(* CODESYS project xlh_ha_client_00_05.project
   Author: Pascal Helfenstein
   Title: xlh_ha
   Company: xemax ag

Project tree, tasks and I/O mapping:
  xlh_base : CODESYS Control for Raspberry Pi 64 SL, CODESYS, order no. 2302000009, version 4.18.0.0
    application app
      libraries: Standard, 3.5.18.0 (System); StringUtils, 3.5.20.0 (System); VisuDialogs, * (System); Web Socket Client SL, 1.12.0.0 (CODESYS); Net Base Services, * (3S - Smart Software Solutions GmbH); MQTT Client SL, 1.12.0.0 (CODESYS); Util, 3.5.21.0 (System); String Functions, * (CODESYS); SysTimeRtc, * (System); SysTime, 3.5.17.0 (System); CmpIecTask, * (System); Memory, 3.5.17.0 (3S - Smart Software Solutions GmbH)
      task MainTask (cyclic, interval t#20ms, priority 1) calls LOCAL_TIME_AND_TIME_ZONE, TASK_INFO, io, MAIN
      task VISU_TASK (cyclic, interval 100 ms, priority 31) calls VisuElems.Visu_Prg
      program MAIN [ST]
      program io [ST]
      IoT/
        DEVICES/
          function block _000_FB_VISU_BASE [ST]
          function block _200_FB_DEVICE_SHELLY_BASE [ST]: statusUpdate, startup, newMessage
          function block _202_FB_DEVICE_SHELLY_1PM_TEMP [ST]: newMessage
          interface IDevice
          interface IDeviceZigbee2Mqtt
          interface IDeviceShelly
          function block _201_FB_DEVICE_SHELLY_1PM_PLUG [ST]: publisher, newMessage
          function block _300_FB_DEVICE_ZIGBEE2MQTT_BASE [ST]: statusUpdate, startup, newMessage
          VISU/
            visualisation VISU_FB_DEVICE_SHELLY_RELAIS
            visualisation VISU_FB_DEVICE_SHELLY_RELAIS_TEMP
          function block _100_FB_DEVICE [ST]: subscriber, publisher, startup, popFifoPublish, newMessage, statusUpdate, pushFifoPublish
          trace Trace (task MainTask): io.fbShellyPlug2._fbMqttPublisher.xBusy, io.fbShellyPlug2._fbMqttPublisher.xDone, io.fbShellyPlug2._fbMqttPublisher.xExecute, io.fbShellyPlug2._iFifoPopCycleCounter
          interface IVisu
        MQTT_Client/
          function TERMINATE_STRING [ST]
          function block FB_MQTT_CLIENT [ST]: pMqttClient
          function GET_VALUE_FROM_MSG [ST]
          function GET_REAL_FROM_VALUE [ST]
          function GET_BOOL_FROM_VALUE [ST]
          function GET_INT_FROM_VALUE [ST]
          function GET_STRING_FROM_VALUE [ST]
          function GET_LREAL_FROM_VALUE [ST]
        global variables GC
        program TASK_INFO [ST]
        program LOCAL_TIME_AND_TIME_ZONE [ST]
      visualisation VISUALIZATION
    SoftMotion General Axis Pool
    GPIOs_A_B : GPIOs A/B, CODESYS, version 4.18.0.0
        unmapped channels: digital inputs (GPIO0..GPIO31), digital outputs (GPIO0..GPIO31)
    Onewire
    Camera device
      <Empty>
    SPI
    I²C
  libraries: VisuSymbols, 4.5.0.0 (System)
  text list GlobalTextList
  5ce3da45-db07-42e7-a21c-a00fff4ed8f6|C:\Users\a.werner\Documents\background.jpg
*)

// xlh_base/app/IoT/GC
{attribute 'qualified_only'}
VAR_GLOBAL CONSTANT
	//STRING_SIZE: INT := 255;
	STRING_SIZE_TOPIC: INT := 1024;
	STRING_SIZE_MESSAGE_TX: INT := 1024;
	STRING_SIZE_MESSAGE_RX: INT := 2048;
END_VAR

// xlh_base/app/IoT/LOCAL_TIME_AND_TIME_ZONE
PROGRAM LOCAL_TIME_AND_TIME_ZONE
VAR_OUTPUT
	stUTC_Timestamp : SysTime;
	stCTE_Timestamp : SysTime;
	stJoinedTimestamp : SysTime;
	stCombinedTimestamp : SysTime;
	uiYear : YEAR; (* 1970..2106 *)
    uiMonth : MONTH;
    uiDay : DAY;
    uiHour : UINT;
    uiMinute : UINT;
    uiSecond : UINT;
    uiMilliseconds : MILLISECOND;
    eWeekday : WEEKDAY;
    datDate : DATE;
    todTime : TIME_OF_DAY;
	eError : Util.ERROR;
	xLeapYear : BOOL;
END_VAR
VAR CONSTANT
    /// Coordinated Universal Time
    gc_tzTimeZoneUTC : TimeZone := (asgPeriod := [(sName:='UTC')]);

    /// Central Europe Time
    gc_tzTimeZoneCET : TimeZone :=
    (
        iBias := 60 (* T#1M => minutes *),
        asgPeriod := [
        ( (* (CEST -> CET) - Last Sunday in Oktober at 03:00:00.000 (CEST) *)
            sName:='CET',
            dtDate := (uiMonth := 10, eWeekday := WEEKDAY.SUNDAY, uiDay := 5, uiHour := 3)
        ),( (* (CET -> CEST) - Last Sunday in March at 02:00:00.000 (CET) *)
            sName := 'CEST',
            dtDate := (uiMonth := 3, eWeekday := WEEKDAY.SUNDAY, uiDay := 5, uiHour := 2),
            iBias := 60 (* T#1M => minutes *)
        )]
    );
END_VAR

SysTimeRtcHighResGet(pTimestamp := stUTC_Timestamp);
// Conversion from UTC timestamp (e.g. from SysTimeRtcHighResGet) to the current period and the local date and time related to the TimeZone parameter.
stCTE_Timestamp := Util.LocalDateTime(	tzTimeZone := gc_tzTimeZoneCET, 
										uliDateTime := stUTC_Timestamp,
										eErrorID => eError);

// Splitting a timestamp into the components of a point in time.
eError := Util.SplitDateTime(	uliDateTime := stCTE_Timestamp,
				uiYear => uiYear,
				uiMonth =>  uiMonth,
				uiDay => uiDay,
				uiHour => uiHour,
				uiMinute => uiMinute,
				uiSecond =>  uiSecond,
				uiMilliseconds => uiMilliseconds,
				eWeekday => eWeekday);

// Joining the components of a point in time to a timestamp (UTC). 
stJoinedTimestamp :=  Util.JoinDateTime( 	uiYear := uiYear,
									uiMonth :=  uiMonth,
									uiDay := uiDay,
									uiHour := uiHour,
									uiMinute := uiMinute,
									uiSecond :=  uiSecond,
									uiMilliseconds := uiMilliseconds);
									
// Separates a timestamp in its IEC data typed parts.
 Util.SeparateDateTime(	uliDateTime := stCTE_Timestamp,
    				eWeekDay => eWeekDay,
    				datDate => datDate,
    				todTime => todTime);
					
// Combines the IEC data typed parts to a timestamp.
stCombinedTimestamp := Util.CombineDateTime(	datDate := datDate, 
												todTime := todTime, 
												eErrorID => eError);
						
// Calculates the appropriate value of the WEEKDAY enum that matches the parameter datDate.
eWeekday := Util.DayOfWeek(	datDate := datDate, 
							eErrorID => eError);

// Checks whether the year (uiYear) passed represents a leap year.					
xLeapYear := Util.IsLeapYear(	uiYear := uiYear,
								eErrorID => eError);

END_PROGRAM

// xlh_base/app/IoT/TASK_INFO
PROGRAM TASK_INFO
VAR
    Result: CmpIecTask.RTS_IEC_RESULT;
    hCurrentTask : CmpIecTask.RTS_IEC_HANDLE;
    pCurrentTaskInfo: POINTER TO Task_Info2;
    stCurrentTaskInfo: Task_Info2;
END_VAR
VAR_OUTPUT
	fCycleTime: LREAL;
	fInterval: LREAL;
	fCycleTimeUs: LREAL;
	fJitterUs: LREAL;
	fJitterOffsetInterwalUs: LREAL;
END_VAR

// https://content.helpme-codesys.com/en/libs/CmpIecTask/Current/index.html
// https://forge.codesys.com/forge/talk/Engineering/thread/b7e9b2b353/
// https://medium.com/@sean.gongz/how-to-get-current-task-actual-cycle-time-in-codesys-267384bcd3b7

hCurrentTask := IecTaskGetCurrent(pResult:=ADR(Result));
pCurrentTaskInfo := IecTaskGetInfo3(hIecTask:=hCurrentTask, pResult:=ADR(Result));
stCurrentTaskInfo := pCurrentTaskInfo^;

fCycleTimeUs := TO_LREAL(TO_DINT(stCurrentTaskInfo.dwInterval) + stCurrentTaskInfo.iJitter);
fInterval := TO_LREAL(stCurrentTaskInfo.dwInterval);
fJitterUs := TO_LREAL(stCurrentTaskInfo.iJitter);
fJitterOffsetInterwalUs := fInterval + fJitterUs;
fCycleTime := fCycleTimeUs / 1000000.0;

END_PROGRAM

// xlh_base/app/io
PROGRAM io
VAR_INPUT
	fbShellyPlug1: _201_FB_DEVICE_SHELLY_1PM_PLUG := (bEnable:=TRUE, sMqttTopicBase:='shellyplug-81', sLabel:='shellyplug-81');
	fbShellyPlug2: _201_FB_DEVICE_SHELLY_1PM_PLUG := (bEnable:=TRUE, sMqttTopicBase:='shellyplug-82', sLabel:='shellyplug-82');
	fbShellyPm1: _201_FB_DEVICE_SHELLY_1PM_PLUG := (bEnable:=FALSE, sMqttTopicBase:='shellyplus1pm-88', sLabel:='shellyplus1pm-88');
	fbShellyPm2: _202_FB_DEVICE_SHELLY_1PM_TEMP := (bEnable:=TRUE, sMqttTopicBase:='shellyplus1pm-51', sLabel:='shellyplus1pm-51');
END_VAR
VAR
	_bStartup: BOOL := TRUE;
	_aIoClients: ARRAY [0..(iNR_OF_IO_CLIENTS-1)] OF POINTER TO _100_FB_DEVICE;
	_fbMqttClient: FB_MQTT_CLIENT := (sClientId:='xlh_base_ha_io');
	_iI: INT;
	//
	_bDummy: BOOL;
END_VAR
VAR CONSTANT
	iNR_OF_IO_CLIENTS: INT := 20;
END_VAR

IF _bStartup THEN
	_bStartup := FALSE;
	_aIoClients[_iI] := ADR(fbShellyPlug1); _iI := _iI + 1;
	_aIoClients[_iI] := ADR(fbShellyPlug2); _iI := _iI + 1;
	_aIoClients[_iI] := ADR(fbShellyPm1); _iI := _iI + 1;
	_aIoClients[_iI] := ADR(fbShellyPm2); _iI := _iI + 1;
	
	FOR _iI := 0 TO (iNR_OF_IO_CLIENTS-1) BY 1 DO
		IF (_aIoClients[_iI] > 16#0) THEN
			_aIoClients[_iI]^.pMqttClient := ADR(_fbMqttClient);
			_aIoClients[_iI]^.startup();	
		END_IF
	END_FOR	
	
	_fbMqttClient.bEnable := TRUE;
END_IF

_fbMqttClient();

FOR _iI := 0 TO (iNR_OF_IO_CLIENTS-1) BY 1 DO
	IF (_aIoClients[_iI] >16#0) THEN
		_aIoClients[_iI]^();	
	END_IF
END_FOR

_bDummy := _fbMqttClient.bConnected;

END_PROGRAM

// xlh_base/app/IoT/DEVICES/_201_FB_DEVICE_SHELLY_1PM_PLUG
FUNCTION_BLOCK _201_FB_DEVICE_SHELLY_1PM_PLUG EXTENDS _200_FB_DEVICE_SHELLY_BASE
VAR_INPUT
	bRelais: BOOL;
	bResetEnergy: BOOL;
END_VAR
VAR_OUTPUT
	bRelaisState: BOOL;
	fVoltage: LREAL;
	fCurrent: LREAL;
	fPower: LREAL;
	fElectricalEnergy: LREAL;
END_VAR
VAR
	//
	_fbRtRelais: R_TRIG;
	_fbFtRelais: F_tRIG;
	_fbTonDiffRelaisState: TON;
END_VAR
VAR CONSTANT
	_tACTION_TIME_NOT_EQUAL: TIME := T#500MS;
END_VAR

SUPER^();
IF bResetEnergy THEN
	fElectricalEnergy := 0.0;
ELSE
	fElectricalEnergy := fElectricalEnergy + fPower * TASK_INFO.fCycleTime;
END_IF

METHOD publisher : BOOL
VAR_INPUT
END_VAR

VAR
	bPublish: BOOL;
	sPublishMessage : STRING(GC.STRING_SIZE_MESSAGE_TX);
END_VAR
THIS^._fbTonDiffRelaisState(IN:=((THIS^.bRelais <> THIS^.bRelaisState) AND NOT _fbTonDiffRelaisState.Q), PT:=THIS^._tACTION_TIME_NOT_EQUAL);
THIS^._fbRtRelais(CLK:=THIS^.bRelais);
THIS^._fbFtRelais(CLK:=THIS^.bRelais);
bPublish := _fbTonDiffRelaisState.Q OR _fbRtRelais.Q OR _fbFtRelais.Q;

IF bPublish THEN
	sPublishMessage := '{"id":1, "src":"';
	Stu.StrConcatA(pstFrom:=ADR(THIS^.sMqttTopicBase), pstTo:=ADR(sPublishMessage), iBufferSize:=GC.STRING_SIZE_MESSAGE_TX);
	Stu.StrConcatA(pstFrom:=ADR('/relais", "method":"Switch.Set", "params":{"id":0, "on":'), pstTo:=ADR(sPublishMessage), iBufferSize:=GC.STRING_SIZE_MESSAGE_TX);
	//sPublishMessage := CONCAT(sPublishMessage, THIS^.sMqttTopicBase);
	//sPublishMessage := CONCAT(sPublishMessage, '/relais", "method":"Switch.Set", "params":{"id":0, "on":');
	IF THIS^.bRelais THEN
		Stu.StrConcatA(pstFrom:=ADR('true}}'), pstTo:=ADR(sPublishMessage), iBufferSize:=GC.STRING_SIZE_MESSAGE_TX);
		//sPublishMessage := CONCAT(sPublishMessage, 'true}}');
	ELSE
		Stu.StrConcatA(pstFrom:=ADR('false}}'), pstTo:=ADR(sPublishMessage), iBufferSize:=GC.STRING_SIZE_MESSAGE_TX);
		//sPublishMessage := CONCAT(sPublishMessage, 'false}}');
	END_IF
	THIS^.pushFifoPublish(THIS^._wsPublishTopic, sPublishMessage);
END_IF

SUPER^.publisher();
END_METHOD

METHOD newMessage : BOOL
VAR_INPUT
	
END_VAR
VAR

	
END_VAR
SUPER^.newMessage();
IF (_fbMqttSubscriber.wsLastTopic = _wsMqttTopicEvent) OR
   (_fbMqttSubscriber.wsLastTopic = _wsMqttTopicStatus) THEN
	bRelaisState := GET_BOOL_FROM_VALUE(bRelaisState, GET_VALUE_FROM_MSG('output', ADR(_sSubscribedMessage)));
	fVoltage := GET_LREAL_FROM_VALUE(fVoltage, GET_VALUE_FROM_MSG('voltage', ADR(_sSubscribedMessage)));
	fCurrent := GET_LREAL_FROM_VALUE(fCurrent, GET_VALUE_FROM_MSG('current', ADR(_sSubscribedMessage)));
	fPower := GET_LREAL_FROM_VALUE(fPower, GET_VALUE_FROM_MSG('apower', ADR(_sSubscribedMessage)));
		
END_IF
IF (_fbMqttSubscriber.wsLastTopic = _wsMqttTopicStatus) THEN
	sSsid := GET_STRING_FROM_VALUE(sSsid, GET_VALUE_FROM_MSG('ssid', ADR(_sSubscribedMessage)));
	sMacId := GET_STRING_FROM_VALUE(sSsid, GET_VALUE_FROM_MSG('bssid', ADR(_sSubscribedMessage)));	
END_IF

(*
// FixMe: total energy from status Message

Topic: shellyplus1pm-51/status/rpcQoS: 0

{"id":1,"src":"shellyplus1pm-e465b8b7ad64","dst":"shellyplus1pm-51/status","result":{"ble":{},"cloud":{"connected":false},"input:0":
{"id":0,"state":false},"mqtt":{"connected":true},
"switch:0":{"id":0, "source":"MQTT", "output":false, "apower":0.0, "voltage":236.0, "current":0.000, 
"aenergy":{"total":2431.000,"by_minute":[0.000,0.000,0.000],"minute_ts":1765258740},
"temperature":{"tC":38.2, "tF":100.8}},"sys":{"mac":"E465B8B7AD64","restart_required":false,"time":"06:39","unixtime":1765258775,"last_sync_ts":1765258399,"uptime":380,"ram_size":250884,"ram_free":138740,"ram_min_free":127852,"fs_size":393216,"fs_free":126976,"cfg_rev":40,"kvs_rev":0,"schedule_rev":1,"webhook_rev":0,"btrelay_rev":0,"available_updates":{},"reset_reason":1,"utc_offset":3600},"temperature:100":{"id": 100,"tC":20.1, "tF":68.1},"temperature:101":{"id": 101,"tC":19.9, "tF":67.9},"temperature:102":{"id": 102,"tC":20.0, "tF":68.0},"wifi":{"sta_ip":"192.168.1.51","status":"got ip","ssid":"hpna_fritz_box","bssid":"3c:37:12:6b:47:96","rssi":-28},"ws":{"connected":false}}}
*)
END_METHOD

END_FUNCTION_BLOCK

// xlh_base/app/IoT/DEVICES/_200_FB_DEVICE_SHELLY_BASE
FUNCTION_BLOCK _200_FB_DEVICE_SHELLY_BASE EXTENDS _100_FB_DEVICE IMPLEMENTS IDeviceShelly
VAR_INPUT
END_VAR
VAR_OUTPUT
	fTemperaturePcb: LREAL;
	sSsid: STRING(255);
	sMacId: STRING(255);
	iRssi: INT;
END_VAR
VAR
	//
	_wsMqttTopicEvent: WSTRING(GC.STRING_SIZE_TOPIC);
	_wsMqttTopicStatus: WSTRING(GC.STRING_SIZE_TOPIC);
	_fTimer: LREAL := 0.0;
END_VAR
VAR CONSTANT
	_fREFRESH_TIME: LREAL := 300.0;
END_VAR

SUPER^();

_fTimer := LIMIT(0.0, _fTimer + TASK_INFO.fCycleTime, 99999.0);
IF _fTimer >= _fREFRESH_TIME THEN
	_fTimer := 0.0;
	statusUpdate();
END_IF

METHOD statusUpdate : BOOL
VAR_INPUT
END_VAR
VAR
	sPublishMessage : STRING(GC.STRING_SIZE_MESSAGE_TX);
END_VAR
SUPER^.statusUpdate();
sPublishMessage := '{"id":1, "src":"';
Stu.StrConcatA(pstFrom:=ADR(THIS^.sMqttTopicBase), pstTo:=ADR(sPublishMessage), iBufferSize:=GC.STRING_SIZE_MESSAGE_TX);
Stu.StrConcatA(pstFrom:=ADR('/status", "method":"Shelly.GetStatus"}'), pstTo:=ADR(sPublishMessage), iBufferSize:=GC.STRING_SIZE_MESSAGE_TX);
//sPublishMessage := CONCAT(sPublishMessage, THIS^.sMqttTopicBase);
//sPublishMessage := CONCAT(sPublishMessage, '/status", "method":"Shelly.GetStatus"}');
THIS^.pushFifoPublish(THIS^._wsPublishTopic, sPublishMessage);
END_METHOD

METHOD startup : BOOL
VAR_INPUT
END_VAR

VAR
END_VAR
SUPER^.startup();

_wsPublishTopic := "";
Stu.StrConcatW(pstFrom:=ADR(_wsMqttTopicBase), pstTo:=ADR(_wsPublishTopic), iBufferSize:=GC.STRING_SIZE_TOPIC);
Stu.StrConcatW(pstFrom:=ADR("/rpc"), pstTo:=ADR(_wsPublishTopic), iBufferSize:=GC.STRING_SIZE_TOPIC);

_wsMqttTopicEvent := "";
Stu.StrConcatW(pstFrom:=ADR(_wsMqttTopicBase), pstTo:=ADR(_wsMqttTopicEvent), iBufferSize:=GC.STRING_SIZE_TOPIC);
Stu.StrConcatW(pstFrom:=ADR("/events/rpc"), pstTo:=ADR(_wsMqttTopicEvent), iBufferSize:=GC.STRING_SIZE_TOPIC);
		
_wsMqttTopicStatus := "";
Stu.StrConcatW(pstFrom:=ADR(_wsMqttTopicBase), pstTo:=ADR(_wsMqttTopicStatus), iBufferSize:=GC.STRING_SIZE_TOPIC);
Stu.StrConcatW(pstFrom:=ADR("/status/rpc"), pstTo:=ADR(_wsMqttTopicStatus), iBufferSize:=GC.STRING_SIZE_TOPIC);
END_METHOD

METHOD newMessage : BOOL
VAR_INPUT
	
END_VAR
VAR

	
END_VAR
SUPER^.newMessage();
IF (_fbMqttSubscriber.wsLastTopic = _wsMqttTopicEvent) OR
   (_fbMqttSubscriber.wsLastTopic = _wsMqttTopicStatus) THEN
   fTemperaturePcb := GET_LREAL_FROM_VALUE(fTemperaturePcb, GET_VALUE_FROM_MSG('temperature":{"tC', ADR(_sSubscribedMessage)));
	iRssi := GET_INT_FROM_VALUE(iRssi, GET_VALUE_FROM_MSG('rssi', ADR(_sSubscribedMessage)));	
END_IF
IF (_fbMqttSubscriber.wsLastTopic = _wsMqttTopicStatus) THEN
	sSsid := GET_STRING_FROM_VALUE(sSsid, GET_VALUE_FROM_MSG('ssid', ADR(_sSubscribedMessage)));
	sMacId := GET_STRING_FROM_VALUE(sSsid, GET_VALUE_FROM_MSG('bssid', ADR(_sSubscribedMessage)));	
END_IF
END_METHOD

END_FUNCTION_BLOCK

// xlh_base/app/IoT/DEVICES/_100_FB_DEVICE
FUNCTION_BLOCK _100_FB_DEVICE EXTENDS _000_FB_VISU_BASE IMPLEMENTS IDevice
VAR_INPUT
	bEnable: BOOL;
	sMqttTopicBase: STRING(255);
	pMqttClient: POINTER TO FB_MQTT_CLIENT;
END_VAR
VAR
	_wsMqttTopicBase: WSTRING(GC.STRING_SIZE_TOPIC);
	//
	_fbRtMqttClientConnected: R_TRIG;
	_fbFtMqttClientConnected: F_TRIG;
	_fbRtMqttSubscriberActive: R_TRIG;
	_fbFtMqttSubscriberActive: F_TRIG;
	_fbRtError: R_TRIG;
	_fbTonConnect: TON;
	_fbTonDisconnect: TON;
	//
	_fbMqttSubscriber : MQTT.MQTTSubscribe;
	_wsSubcribedTopicFilter : WSTRING(GC.STRING_SIZE_TOPIC);
	_sSubscribedMessage : STRING(GC.STRING_SIZE_MESSAGE_RX);	
	//
	_fbMqttPublisher : MQTT.MQTTPublish;
	_wsPublishTopic : WSTRING(GC.STRING_SIZE_TOPIC);
	_sPublishMessage : STRING(GC.STRING_SIZE_MESSAGE_TX);
	//
	_iFifoPos: INT;
	_iFifoPosMax: INT;
	_awsPublishTopic: ARRAY[0..(_iFIFO_SIZE-1)] OF WSTRING(GC.STRING_SIZE_TOPIC);
	_asPublishMessage: ARRAY[0..(_iFIFO_SIZE-1)] OF STRING(GC.STRING_SIZE_MESSAGE_TX);
	_iFifoPopCycleCounter: INT;
	//
	_todMessageUpdate: TIME_OF_DAY;
END_VAR
VAR CONSTANT
	_iFIFO_SIZE: INT := 25;
	_iFIFO_DELAY_COUNTER: INT := 5;
END_VAR

THIS^.subscriber();
THIS^.publisher();

METHOD subscriber : BOOL
VAR_INPUT
END_VAR
THIS^._fbRtMqttClientConnected(CLK:=THIS^.pMqttClient^.bConnected);
THIS^._fbFtMqttClientConnected(CLK:=THIS^.pMqttClient^.bConnected);
THIS^._fbRtError(CLK:=THIS^.pMqttClient^.bError);
IF THIS^._fbRtMqttClientConnected.Q THEN
	THIS^._fbMqttSubscriber.xEnable := TRUE;
END_IF
IF THIS^._fbRtError.Q OR THIS^._fbFtMqttClientConnected.Q THEN
	THIS^._fbMqttSubscriber.xEnable := FALSE;
END_IF
THIS^._fbTonDisconnect.IN := THIS^.pMqttClient^.bConnected AND THIS^._fbMqttSubscriber.xEnable AND NOT THIS^._fbMqttSubscriber.xBusy;
THIS^._fbTonDisconnect(PT:=T#3000MS);
IF THIS^._fbTonDisconnect.Q THEN
	THIS^._fbMqttSubscriber.xEnable := FALSE;
END_IF
THIS^._fbTonConnect.IN := THIS^.pMqttClient^.bConnected AND NOT THIS^._fbMqttSubscriber.xEnable;
THIS^._fbTonConnect(PT:=T#500MS);
IF THIS^._fbTonConnect.Q THEN
	THIS^._fbMqttSubscriber.xEnable := TRUE;
END_IF
IF NOT THIS^.bEnable THEN
	THIS^._fbMqttSubscriber.xEnable := FALSE;
END_IF

THIS^._fbMqttSubscriber(mqttClient:=THIS^.pMqttClient^.fbMqttClient,
				wsTopicFilter:=THIS^._wsSubcribedTopicFilter,
		        pbPayload:=ADR(THIS^._sSubscribedMessage),
				udiMaxPayloadSize:=SIZEOF(THIS^._sSubscribedMessage));
TERMINATE_STRING(psIn:=ADR(THIS^._sSubscribedMessage), THIS^._fbMqttSubscriber.udiPayloadSize);

IF THIS^._fbMqttSubscriber.xReceived THEN
	THIS^.newMessage();
END_IF 

THIS^._fbRtMqttSubscriberActive(CLK:=THIS^._fbMqttSubscriber.xSubscribeActive);
THIS^._fbFtMqttSubscriberActive(CLK:=THIS^._fbMqttSubscriber.xSubscribeActive);
IF THIS^._fbRtMqttSubscriberActive.Q THEN
	THIS^.statusUpdate();
END_IF
			
_bDummy := THIS^._fbMqttSubscriber.xEnable;				
_bDummy := THIS^._fbMqttSubscriber.xDone;
_bDummy := THIS^._fbMqttSubscriber.xBusy;
_bDummy := THIS^._fbMqttSubscriber.xError;
_bDummy := THIS^._fbMqttSubscriber.xSubscribeActive;
_wsDummy := THIS^._fbMqttSubscriber.wsLastTopic;
_sDummy := THIS^._sSubscribedMessage;
END_METHOD

METHOD publisher : BOOL
VAR_INPUT

END_VAR
IF THIS^.bEnable THEN
	IF NOT THIS^._fbMqttPublisher.xExecute AND NOT THIS^._fbMqttPublisher.xBusy  THEN
		THIS^._fbMqttPublisher.xExecute := popFifoPublish();  
	END_IF
ELSE
	THIS^._fbMqttPublisher.xExecute := FALSE;
END_IF

THIS^._fbMqttPublisher(mqttClient:=THIS^.pMqttClient^.fbMqttClient, 	 
					   wsTopicName:=_wsPublishTopic,
					   udiTimeOut:=10000,
					   pbPayload:=ADR(_sPublishMessage),
					   udiPayloadSize:=DINT_TO_UDINT(Stu.StrLenA(ADR(_sPublishMessage))));

IF NOT THIS^._fbMqttPublisher.xBusy or THIS^._fbMqttPublisher.xError THEN
	THIS^._fbMqttPublisher.xExecute := FALSE;  
END_IF
END_METHOD

METHOD startup : BOOL
VAR_INPUT
END_VAR

VAR
END_VAR
_wsMqttTopicBase := STRING_TO_WSTRING(sMqttTopicBase);

_wsSubcribedTopicFilter := "";
Stu.StrConcatW(pstFrom:=ADR(_wsMqttTopicBase), pstTo:=ADR(_wsSubcribedTopicFilter), iBufferSize:=GC.STRING_SIZE_TOPIC);
Stu.StrConcatW(pstFrom:=ADR("/#"), pstTo:=ADR(_wsSubcribedTopicFilter), iBufferSize:=GC.STRING_SIZE_TOPIC);
END_METHOD

METHOD popFifoPublish : BOOL
VAR_INPUT

END_VAR
VAR
	iI: INT;
END_VAR
IF _iFifoPos > 0  AND _iFifoPopCycleCounter = 0 THEN
	_iFifoPos := _iFifoPos - 1;
	//MEM.MemFill(ADR(sPublishTopic), INT_TO_UINT(SIZEOF(sPublishTopic)), 16#00);
	//MEM.MemFill(ADR(sPublishMessage), INT_TO_UINT(SIZEOF(sPublishMessage)), 16#00);	
	MEM.MemMove(ADR(_awsPublishTopic[0]), ADR(_wsPublishTopic), SIZEOF(_wsPublishTopic));
	MEM.MemMove(ADR(_asPublishMessage[0]), ADR(_sPublishMessage), SIZEOF(_sPublishMessage));
	FOR iI := 1 TO (_iFIFO_SIZE-1) BY 1 DO
		MEM.MemMove(ADR(_awsPublishTopic[iI]), ADR(_awsPublishTopic[iI-1]), SIZEOF(_awsPublishTopic[iI-1]));
		MEM.MemMove(ADR(_asPublishMessage[iI]), ADR(_asPublishMessage[iI-1]), SIZEOF(_asPublishMessage[iI-1]));
	END_FOR 
	MEM.MemFill(ADR(_awsPublishTopic[_iFIFO_SIZE-1]), SIZEOF(_awsPublishTopic[_iFIFO_SIZE-1]), 16#00);
	MEM.MemFill(ADR(_asPublishMessage[_iFIFO_SIZE-1]), SIZEOF(_asPublishMessage[_iFIFO_SIZE-1]), 16#00);
	
	_iFifoPopCycleCounter := _iFIFO_DELAY_COUNTER;
	popFifoPublish := TRUE;
ELSE
	IF _iFifoPopCycleCounter > 0 THEN
		_iFifoPopCycleCounter := _iFifoPopCycleCounter - 1;
	END_IF
	popFifoPublish := FALSE;	
END_IF
END_METHOD

METHOD newMessage : BOOL
VAR_INPUT
	
END_VAR
VAR

	
END_VAR
THIS^._todMessageUpdate := LOCAL_TIME_AND_TIME_ZONE.todTime;
END_METHOD

METHOD statusUpdate : BOOL
VAR_INPUT
END_VAR

VAR
END_VAR
END_METHOD

METHOD pushFifoPublish : BOOL
VAR_INPUT
	wsTopic: WSTRING(GC.STRING_SIZE_TOPIC);
	sMessage: STRING(GC.STRING_SIZE_MESSAGE_TX);
END_VAR
VAR
	iI: INT;
END_VAR
IF THIS^.bEnable AND _iFifoPos < (_iFIFO_SIZE-1) THEN
	_iFifoPos := _iFifoPos + 1;
	FOR iI := (_iFIFO_SIZE-2) TO 0 BY -1 DO
		MEM.MemMove(ADR(_awsPublishTopic[iI]), ADR(_awsPublishTopic[iI+1]), SIZEOF(_awsPublishTopic[iI+1]));
		MEM.MemMove(ADR(_asPublishMessage[iI]), ADR(_asPublishMessage[iI+1]), SIZEOF(_asPublishMessage[iI+1]));
	END_FOR 
	MEM.MemFill(ADR(_awsPublishTopic[0]), SIZEOF(_awsPublishTopic[0]), 16#00);
	MEM.MemMove(ADR(wsTopic), ADR(_awsPublishTopic[0]), SIZEOF(wsTopic));
	TERMINATE_STRING(psIn:=ADR(_awsPublishTopic[0]), udiLength:=SIZEOF(wsTopic)-1);
	
	MEM.MemFill(ADR(_asPublishMessage[0]), SIZEOF(_asPublishMessage[0]), 16#00);
	MEM.MemMove(ADR(sMessage), ADR(_asPublishMessage[0]), SIZEOF(sMessage));
	TERMINATE_STRING(psIn:=ADR(_asPublishMessage[0]), udiLength:=SIZEOF(sMessage)-1);
	
	pushFifoPublish := TRUE;
ELSE
	pushFifoPublish := FALSE;	
END_IF

IF _iFifoPos > _iFifoPosMax THEN
	_iFifoPosMax := _iFifoPos;
END_IF
END_METHOD

END_FUNCTION_BLOCK

// xlh_base/app/IoT/DEVICES/_000_FB_VISU_BASE
FUNCTION_BLOCK _000_FB_VISU_BASE IMPLEMENTS IVisu
VAR_INPUT
	sLabel: STRING(255) := '';
END_VAR
VAR
	//_bVisuFramShow: BOOL;
	//_iVisuFrame: INT;	
	//_tonVisuFrameShow: TON;
	_bDummy: BOOL;
	_iDummy: INT;
	_rDummy: REAL;
	_fDummy: LREAL;
	_sDummy: STRING(GC.STRING_SIZE_MESSAGE_RX);
	_wsDummy: WSTRING(GC.STRING_SIZE_TOPIC);
END_VAR

(*
_tonVisuFrameShow(IN:=_bVisuFramShow, PT:=T#300S);
IF _tonVisuFrameShow.Q THEN
	_bVisuFramShow := FALSE;
	_iVisuFrame := 0;
END_IF
*)

END_FUNCTION_BLOCK

// xlh_base/app/IoT/DEVICES/IVisu
INTERFACE IVisu

END_INTERFACE

// xlh_base/app/IoT/DEVICES/IDevice
INTERFACE IDevice

END_INTERFACE

// xlh_base/app/IoT/MQTT_Client/FB_MQTT_CLIENT
FUNCTION_BLOCK FB_MQTT_CLIENT
VAR_INPUT
	bEnable: BOOL;
	sHostname: STRING(255) := 'localhost';	
	sClientId: STRING(255) := 'xLH_mqtt_codesys';	
END_VAR
VAR_OUTPUT
	bConnected: BOOL;
	bError: BOOL;
	fbMqttClient : MQTT.MQTTClient := (uiPort:=1883, eMQTTVersion:=MQTT.MQTT_VERSION.V3_1_1, eCommunicationMode:= MQTT.COMMUNICATION_MODE.TCP);
END_VAR
VAR
	_refMqttClient: REFERENCE TO MQTT.MQTTClient;
	_bStartup: BOOL := TRUE;
END_VAR

IF _bStartup THEN
	_bStartup := FALSE;
	_refMqttClient REF= fbMqttClient;
END_IF
fbMqttClient.xEnable := bEnable AND NOT fbMqttClient.xError;
fbMqttClient.sClientId := sClientId;
fbMqttClient(sHostname:=sHostname);
bConnected := fbMqttClient.xConnectedToBroker;
bError := fbMqttClient.xError;

PROPERTY pMqttClient : POINTER TO FB_MQTT_CLIENT
GET
pMqttClient := ADR(THIS^.fbMqttClient);
END_GET
END_PROPERTY

END_FUNCTION_BLOCK

// xlh_base/app/IoT/MQTT_Client/TERMINATE_STRING
// Terminates the STRING psIn at position udiLength
FUNCTION TERMINATE_STRING : BOOL
VAR_INPUT
	psIn : POINTER TO BYTE; // Pointer to STRING
	udiLength : UDINT; // Length of psIn
END_VAR
VAR
END_VAR

psIn[udiLength] := 0;
TERMINATE_STRING := TRUE;

END_FUNCTION

// xlh_base/app/IoT/DEVICES/IDeviceShelly
INTERFACE IDeviceShelly

END_INTERFACE

// xlh_base/app/IoT/MQTT_Client/GET_LREAL_FROM_VALUE
FUNCTION GET_LREAL_FROM_VALUE: LREAL;
VAR_INPUT
	fValue: LREAL;
	sValue: STRING(255);
END_VAR

IF sValue <> '' THEN
	fValue := STRING_TO_LREAL(sValue);
END_IF
GET_LREAL_FROM_VALUE := fValue;

END_FUNCTION

// xlh_base/app/IoT/MQTT_Client/GET_VALUE_FROM_MSG
FUNCTION GET_VALUE_FROM_MSG: STRING(255)
VAR_INPUT
	sKey: STRING(255);
	pSubscribedMessage: POINTER TO STRING(GC.STRING_SIZE_MESSAGE_RX);
END_VAR
VAR
	iStrFindPos1: INT;
	iStrFindPos2: INT;
	sMessage : STRING(255);
	sValue : STRING(255);
END_VAR

sKey := CONCAT(CONCAT('"', sKey), '":'); 		

iStrFindPos1 := MAX(0, Stu.StrFindA(pst1:=pSubscribedMessage, pst2:=ADR(sKey), uiSearchStart:=0));
Stu.StrCpyA(pBuffer:=ADR(sMessage), 
			iBufferSize:=SIZEOF(sMessage)-50, 
			pStr:=pSubscribedMessage+INT_TO_DWORD(iStrFindPos1));  

iStrFindPos1 := MAX(0, Stu.StrFindA(pst1:=ADR(sMessage), 
                                    pst2:=ADR(':'), 
                                    uiSearchStart:=INT_TO_UINT(MAX(0, LEN(sKey)-1))));		 
iStrFindPos2 := MAX(0, Stu.StrFindA(pst1:=ADR(sMessage), 
                                    pst2:=ADR(','), 
                                    uiSearchStart:=INT_TO_UINT(MAX(0, LEN(sKey)))));		
IF iStrFindPos2 = 0 THEN
	iStrFindPos2 := MAX(0, Stu.StrFindA(pst1:=ADR(sMessage), 
                                    pst2:=ADR('}'), 
                                    uiSearchStart:=INT_TO_UINT(MAX(0, LEN(sKey)))));
END_IF
// Falls das Property nicht vorhanden ist, keine Aenderung (MID, LEFT funktionieren nur bei Zeichenketten len < 255)
IF (iStrFindPos1 <> 0) AND (iStrFindPos2 <> 0) THEN
	sValue := MID(sMessage, iStrFindPos2-iStrFindPos1-1, iStrFindPos1+1);
	// bei einem String sind die " zu enternen
	IF LEFT(sMessage, 1) = '"' THEN
		sValue := MID(sValue, LEN(sValue)-2, 2);
	END_IF
ELSE
	sValue := '';
END_IF
		
(*
sValue := '';
sValue := CONCAT(sValue, INT_TO_STRING(iStrFindPos1));
sValue := CONCAT(sValue, ' | ');
sValue := CONCAT(sValue, INT_TO_STRING(iStrFindPos2));
sValue := CONCAT(sValue, ' | ');
sValue := CONCAT(sValue, sMessage);
*)

GET_VALUE_FROM_MSG := sValue;

END_FUNCTION

// xlh_base/app/IoT/MQTT_Client/GET_INT_FROM_VALUE
FUNCTION GET_INT_FROM_VALUE: INT;
VAR_INPUT
	iValue: int;
	sValue: STRING(255);
END_VAR

IF sValue <> '' THEN
	iValue := STRING_TO_INT(sValue);
END_IF
GET_INT_FROM_VALUE := iValue;

END_FUNCTION

// xlh_base/app/IoT/MQTT_Client/GET_STRING_FROM_VALUE
FUNCTION GET_STRING_FROM_VALUE: STRING(255);
VAR_INPUT
	_sValue: STRING(255);
	sValue: STRING(255);
END_VAR

IF sValue <> '' THEN
	_sValue := sValue;
END_IF
GET_STRING_FROM_VALUE := _sValue;

END_FUNCTION

// xlh_base/app/IoT/MQTT_Client/GET_BOOL_FROM_VALUE
FUNCTION GET_BOOL_FROM_VALUE: BOOL;
VAR_INPUT
	bValue: BOOL;
	sValue: STRING(255);
END_VAR

IF sValue <> '' THEN
	bValue := (sValue = 'true');
END_IF
GET_BOOL_FROM_VALUE := bValue;

END_FUNCTION

// xlh_base/app/IoT/DEVICES/_202_FB_DEVICE_SHELLY_1PM_TEMP
FUNCTION_BLOCK _202_FB_DEVICE_SHELLY_1PM_TEMP EXTENDS _201_FB_DEVICE_SHELLY_1PM_PLUG
VAR_OUTPUT
	fTemperature1: LREAL;
	fTemperature2: LREAL;
	fTemperature3: LREAL;
	fTemperatureMean: LREAL;
END_VAR

SUPER^();
fTemperatureMean := (fTemperature1+fTemperature2+fTemperature3)/3.0;

METHOD newMessage : BOOL
VAR_INPUT
	
END_VAR
VAR

	
END_VAR
SUPER^.newMessage();
IF (_fbMqttSubscriber.wsLastTopic = _wsMqttTopicEvent) OR
   (_fbMqttSubscriber.wsLastTopic = _wsMqttTopicStatus) THEN
	fTemperature1 := GET_LREAL_FROM_VALUE(fTemperature1, GET_VALUE_FROM_MSG('temperature:100":{"id": 100,"tC', ADR(_sSubscribedMessage)));
	fTemperature1 := GET_LREAL_FROM_VALUE(fTemperature1, GET_VALUE_FROM_MSG('temperature:100":{"tC', ADR(_sSubscribedMessage)));
	fTemperature2 := GET_LREAL_FROM_VALUE(fTemperature2, GET_VALUE_FROM_MSG('temperature:101":{"id": 101,"tC', ADR(_sSubscribedMessage)));
	fTemperature2 := GET_LREAL_FROM_VALUE(fTemperature2, GET_VALUE_FROM_MSG('temperature:101":{"tC', ADR(_sSubscribedMessage)));
	fTemperature3 := GET_LREAL_FROM_VALUE(fTemperature3, GET_VALUE_FROM_MSG('temperature:102":{"id": 102,"tC', ADR(_sSubscribedMessage)));
	fTemperature3 := GET_LREAL_FROM_VALUE(fTemperature3, GET_VALUE_FROM_MSG('temperature:102":{"tC', ADR(_sSubscribedMessage)));
END_IF
END_METHOD

END_FUNCTION_BLOCK

// xlh_base/app/MAIN
PROGRAM MAIN
VAR
END_VAR

(*
IP Shelly Accesspoint: 192.168.33.1
FixMe:
- Publisher Stu Bibliothek anstelle Standardstringoperationen (len < 255);
- Dokumentation IoT Code
*)

END_PROGRAM

// xlh_base/app/IoT/MQTT_Client/GET_REAL_FROM_VALUE
FUNCTION GET_REAL_FROM_VALUE: REAL;
VAR_INPUT
	rValue: REAL;
	sValue: STRING(255);
END_VAR

IF sValue <> '' THEN
	rValue := STRING_TO_LREAL(sValue);
END_IF
GET_REAL_FROM_VALUE := rValue;

END_FUNCTION

// xlh_base/app/IoT/DEVICES/IDeviceZigbee2Mqtt
INTERFACE IDeviceZigbee2Mqtt

END_INTERFACE

// xlh_base/app/IoT/DEVICES/_300_FB_DEVICE_ZIGBEE2MQTT_BASE
FUNCTION_BLOCK _300_FB_DEVICE_ZIGBEE2MQTT_BASE EXTENDS _100_FB_DEVICE IMPLEMENTS IDeviceShelly
VAR_INPUT
END_VAR
VAR_OUTPUT
	rTemperaturePcb: REAL;
	sSsid: STRING(255);
	sMacId: STRING(255);
	iRssi: INT;
END_VAR
VAR
	//
	_wsMqttTopicEvent: WSTRING(GC.STRING_SIZE_TOPIC) := "shellyplus-51/status/rpc";
	_wsMqttTopicStatus: WSTRING(GC.STRING_SIZE_TOPIC) := "shellyplus-51/status/rpc";
	_rTimer: REAL := 0.0;
END_VAR
VAR CONSTANT
	_rREFRESH_TIME: REAL := 300.0;
END_VAR

SUPER^();

_rTimer := LIMIT(0.0, _rTimer + TASK_INFO.fCycleTime, 99999.0);
IF _rTimer >= _rREFRESH_TIME THEN
	_rTimer := 0.0;
	statusUpdate();
END_IF

METHOD statusUpdate : BOOL
VAR_INPUT
END_VAR

VAR
END_VAR
SUPER^.statusUpdate();

THIS^._fbMqttPublisher.xExecute := TRUE;
THIS^._sPublishMessage := '{"id":1, "src":"';
THIS^._sPublishMessage := CONCAT(THIS^._sPublishMessage, THIS^._sMqttTopicBase);
THIS^._sPublishMessage := CONCAT(THIS^._sPublishMessage, '/status", "method":"Shelly.GetStatus"}');

// '{"id":1, "src":"shellyplus-51/status", "method":"Shelly.GetStatus"}'
END_METHOD

METHOD startup : BOOL
VAR_INPUT
END_VAR

VAR
END_VAR
SUPER^.startup();

_wsMqttTopicEvent := "";
Stu.StrConcatW(pstFrom:=ADR(_wsMqttTopicBase), pstTo:=ADR(_wsMqttTopicEvent), iBufferSize:=GC.STRING_SIZE_TOPIC);
Stu.StrConcatW(pstFrom:=ADR("/events/rpc"), pstTo:=ADR(_wsMqttTopicEvent), iBufferSize:=GC.STRING_SIZE_TOPIC);
		
_wsMqttTopicStatus := "";
Stu.StrConcatW(pstFrom:=ADR(_wsMqttTopicBase), pstTo:=ADR(_wsMqttTopicStatus), iBufferSize:=GC.STRING_SIZE_TOPIC);
Stu.StrConcatW(pstFrom:=ADR("/status/rpc"), pstTo:=ADR(_wsMqttTopicStatus), iBufferSize:=GC.STRING_SIZE_TOPIC);
END_METHOD

METHOD newMessage : BOOL
VAR_INPUT
	
END_VAR
VAR

	
END_VAR
SUPER^.newMessage();
IF (_fbMqttSubscriber.wsLastTopic = _wsMqttTopicEvent) OR
   (_fbMqttSubscriber.wsLastTopic = _wsMqttTopicStatus) THEN
   rTemperaturePcb := GET_REAL_FROM_VALUE(rTemperaturePcb, GET_VALUE_FROM_MSG('temperature":{"tC', ADR(_sSubscribedMessage)));
	iRssi := GET_INT_FROM_VALUE(iRssi, GET_VALUE_FROM_MSG('rssi', ADR(_sSubscribedMessage)));	
END_IF
IF (_fbMqttSubscriber.wsLastTopic = _wsMqttTopicStatus) THEN
	sSsid := GET_STRING_FROM_VALUE(sSsid, GET_VALUE_FROM_MSG('ssid', ADR(_sSubscribedMessage)));
	sMacId := GET_STRING_FROM_VALUE(sSsid, GET_VALUE_FROM_MSG('bssid', ADR(_sSubscribedMessage)));	
END_IF
END_METHOD

END_FUNCTION_BLOCK

// xlh_base/app/IoT/DEVICES/VISU/VISU_FB_DEVICE_SHELLY_RELAIS
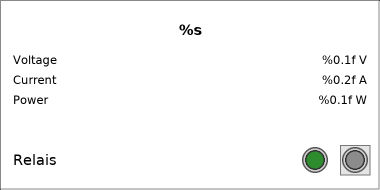
VISUALIZATION VISU_FB_DEVICE_SHELLY_RELAIS  // 380x190
VAR_INPUT
   {attribute 'parameterstringof' := 'fbDevice'}
   sFbInstanceName : STRING;
END_VAR
VAR_IN_OUT
   fbDevice: _201_FB_DEVICE_SHELLY_1PM_PLUG;
END_VAR
    Rectangle (0,0 381x191)
    Rectangle (10,140 281x40), "Relais"
    Rectangle (10,10 361x40), "%s", text variable: fbDevice.sLabel
    Lamp1 (300,140 30x40), variable: fbDevice.bRelaisState, style: Lamp-Lamp1-Green
    PushSwitch (340,140 30x40), variable: fbDevice.bRelais, behaviour: TOGGLE, style: Switch-PushSwitch-Gray
    Rectangle (10,50 261x20), "Voltage"
    Rectangle (270,50 100x20), "%0.1f V", text variable: fbDevice.fVoltage
    Rectangle (270,70 100x20), "%0.2f A", text variable: fbDevice.fCurrent
    Rectangle (10,70 261x20), "Current"
    Rectangle (270,90 100x20), "%0.1f W", text variable: fbDevice.fPower
    Rectangle (10,90 261x20), "Power"
END_VISUALIZATION

// xlh_base/app/VISUALIZATION
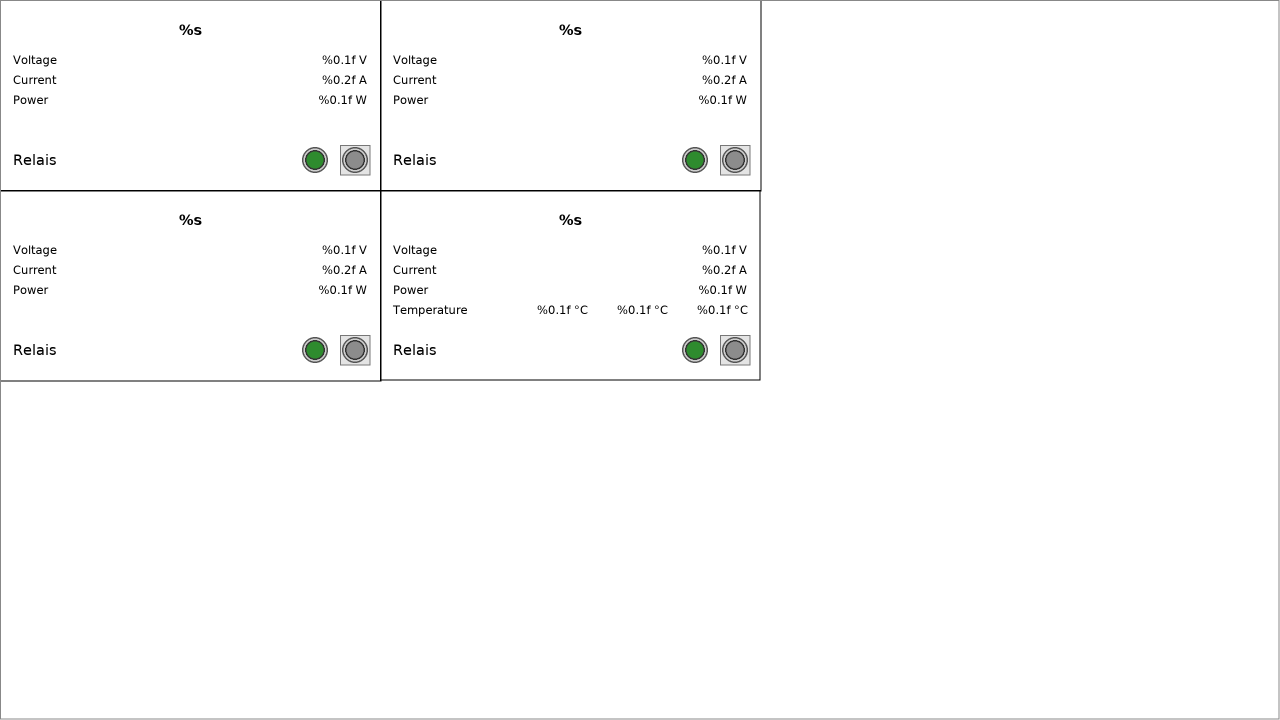
VISUALIZATION VISUALIZATION  // 1280x720
    Frame (0,0 380x191)
        shows VISU_FB_DEVICE_SHELLY_RELAIS(fbDevice := io.fbShellyPlug1)
    Frame (380,0 380x191)
        shows VISU_FB_DEVICE_SHELLY_RELAIS(fbDevice := io.fbShellyPlug2)
    Frame (0,190 380x191)
        shows VISU_FB_DEVICE_SHELLY_RELAIS(fbDevice := io.fbShellyPm1)
    Frame (380,190 380x191)
        shows VISU_FB_DEVICE_SHELLY_RELAIS_TEMP(fbDevice := io.fbShellyPm2)
END_VISUALIZATION

// xlh_base/app/IoT/DEVICES/VISU/VISU_FB_DEVICE_SHELLY_RELAIS_TEMP
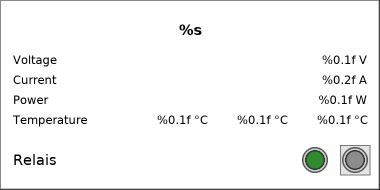
VISUALIZATION VISU_FB_DEVICE_SHELLY_RELAIS_TEMP  // 380x190
VAR_INPUT
   {attribute 'parameterstringof' := 'fbDevice'}
   sFbInstanceName : STRING;
END_VAR
VAR_IN_OUT
   fbDevice: _202_FB_DEVICE_SHELLY_1PM_TEMP;
END_VAR
    Rectangle (0,0 380x190)
    Rectangle (10,140 281x40), "Relais"
    Rectangle (10,10 361x40), "%s", text variable: fbDevice.sLabel
    Lamp1 (300,140 30x40), variable: fbDevice.bRelaisState, style: Lamp-Lamp1-Green
    PushSwitch (340,140 30x40), variable: fbDevice.bRelais, behaviour: TOGGLE, style: Switch-PushSwitch-Gray
    Rectangle (10,50 261x20), "Voltage"
    Rectangle (270,50 100x20), "%0.1f V", text variable: fbDevice.fVoltage
    Rectangle (270,70 100x20), "%0.2f A", text variable: fbDevice.fCurrent
    Rectangle (10,70 261x20), "Current"
    Rectangle (270,90 100x20), "%0.1f W", text variable: fbDevice.fPower
    Rectangle (10,90 261x20), "Power"
    Rectangle (10,110 111x20), "Temperature"
    Rectangle (210,110 81x20), "%0.1f °C", text variable: fbDevice.fTemperature2
    Rectangle (290,110 81x20), "%0.1f °C", text variable: fbDevice.fTemperature3
    Rectangle (130,110 81x20), "%0.1f °C", text variable: fbDevice.fTemperature1
END_VISUALIZATION
